RESOURCE_TYPE TestResource
  FB_TYPES
    TEST_START_FB;
  END_FB_TYPES
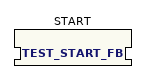
  FBS
    START : TEST_START_FB;
  END_FBS
END_RESOURCE_TYPE
